FUNCTION_BLOCK FB_RefDummy
VAR_INPUT
	input_6  :BOOL;

	input_1  :BOOL;
    input_2  :BOOL;
    input_3  :BOOL;
    input_4  :BOOL;
    input_5  :BOOL;
    
END_VAR
VAR_OUTPUT

	output_1  :BOOL;
    output_2  :BOOL;
    output_3  :BOOL;

END_VAR
VAR
END_VAR

// NETWORK 1

END_FUNCTION_BLOCK

(* stored: Version 1.1.0.1, ProductVersion 3.1.4024.12
   POU FB_RefDummy: Id {26f3df04-2c37-459f-bbef-39642d3b4525}, SpecialFunc None *)
